FUNCTION_BLOCK EL1809
VAR
	_io : EL1xx9_Data;
	{attribute addProperty Name "WcState"}
	_wcState : WcStateInputToggle;
	{attribute addProperty Name "Info data"}
	_infoData : InfoDataBase;
END_VAR

PROPERTY IO : REFERENCE TO EL1xx9_Data
GET
IO REF= _io;
END_GET
END_PROPERTY

PROPERTY WcState : REFERENCE TO WcStateInputToggle
GET
WcState REF= _wcState;
END_GET
END_PROPERTY

END_FUNCTION_BLOCK

(* stored: Version 1.1.0.1, ProductVersion 3.1.4024.9
   POU EL1809: Id {4067506e-2852-0893-1edb-5fd46d2c9b67}, SpecialFunc None
   Property IO: Id {415dd3a3-b86b-0eec-0e7d-d787d2620359}
   Get Get: Id {a493393d-bdfc-0184-390d-63ea75ea9ac2}
   Property WcState: Id {a69a8bc8-4cba-082c-320a-349eec7066a2}
   Get Get: Id {cbfa59ec-71a9-03a3-2431-013c45d94bc0} *)
